// TIA Portal V17 export
// export: Created 2024-09-02T12:50:31.0700232Z, ExportSetting WithDefaults, DisplayName Totally Integrated Automation Portal, DisplayVersion V17, DisplayName TIA Portal Openness, DisplayVersion V17, DisplayName TIA Portal Version Control Interface, DisplayVersion V17, DisplayName STEP 7 Professional, DisplayVersion V17, DisplayName STEP 7 Safety, DisplayVersion V17, DisplayName WinCC Professional, DisplayVersion V17
TYPE "Desoutter_Output"
// stored: IsFailsafeCompliant false
   STRUCT
      Accept_Report : Bool;   // Active when the cycle is over and the tightening cycle report is OK.
      Reject_Report : Bool;   // Active when the cycle is over and the tightening cycle report is NOK.
      Number_of_cycles_OK : Bool;   // This signal switches to “1” when the number of cycles run with an Accept Report is equal to the programmed number of cycles OK in the selected cycle parameters.
      In_Cycle : Bool;   // Response to the Start Cycle request. Drops to “0” at the end of a tightening or untightening.
      Ready : Bool;   // This signal is at “1” when the controller is in working order.
      Run_reverse_enabled : Bool;   // A spindle Reverse validation has been activated.
      Synchro_OUT : Bool;   // Used in conjunction with Synchro IN input to synchronise the tightening cycle phases of several controllers (synchro waiting phase).
      CycleEcho : Byte;   // Binary coded 1-2-4-8 selected cycle echo. The cycle echo is sent back only if it corresponds to a programmed cycle in the station. Otherwise it is at “0”.
      Result : Struct
         "Torque Result" : Real;   // this is the IEEE float value of the torque displayed on the controller.
         "Torque Trend" : Int;   // 0x00 No report, 0x01 Torque is below the lower limit, 0x02 Torque is over the upper limit, 0x03 Torque is in the limits
         "Angle Result" : Real;   // this is the IEEE float value of the angle displayed on the controller.
         "Angle Trend" : Int;   // 0x00 No report,0x01 Angle is below the lower limit,0x02 Angle is over the upper limit,0x03 Angle is in the limits
      END_STRUCT;
      "PART _ID" : Array[1..32] of Char;   // Part numer
   END_STRUCT;
END_TYPE
